FUNCTION_BLOCK MMotor
VAR_INPUT
	start AT %I* : BOOL;
	stop AT %I* : BOOL; 
END_VAR
VAR_OUTPUT
	motor AT %Q* : BOOL;
END_VAR
VAR
END_VAR

IF start THEN
	motor := TRUE;
ELSIF stop THEN
	motor := FALSE;
END_IF

END_FUNCTION_BLOCK

(* stored: Version 1.1.0.1
   POU MMotor: Id {e442abd9-743e-4cf6-afd8-dd06585db08a}, SpecialFunc None *)
